INTERFACE Disposable EXTENDS Queryable

METHOD Dispose
END_METHOD

END_INTERFACE

(* stored: Version 1.1.0.1
   Itf Disposable: Id {686d83f0-17e8-0722-3054-7fbae1a1792f}
   Method Dispose: Id {a1bd5f5a-1aeb-083f-3439-f3c8e4cb69f4} *)
